FUNCTION_BLOCK Moto1 EXTENDS Vehiculo
VAR_INPUT
	Aceleracion : REAL;
END_VAR
VAR_OUTPUT
END_VAR
VAR
END_VAR


METHOD Mover : REAL
VAR_INPUT
	Velocidad_Deseada : REAL;
END_VAR
Mover := Velocidad_Deseada * Aceleracion ;
END_METHOD

END_FUNCTION_BLOCK

(* stored: Version 1.1.0.1, ProductVersion 3.1.4024.12
   POU Moto1: Id {3ad43376-49ab-444b-a93a-f983711d4a1e}, SpecialFunc None
   Method Mover: Id {f6b9738a-e6e2-49b6-8dfb-d1e036957184} *)
